FUNCTION_BLOCK STATE_LOGGER_SIMPLE
  {SET_ATTRIBUTE(OpcUa, SERVICE)}
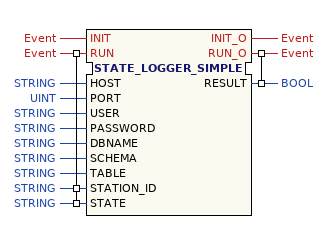
  EVENT_INPUT
    INIT;
    RUN WITH STATION_ID, STATE;
  END_EVENT
  EVENT_OUTPUT
    INIT_O;
    RUN_O WITH RESULT;
  END_EVENT
  VAR_INPUT
    HOST : STRING;
    PORT : UINT;
    USER : STRING;
    PASSWORD : STRING;
    DBNAME : STRING;
    SCHEMA : STRING;
    TABLE : STRING;
    STATION_ID : STRING;
    STATE : STRING;
  END_VAR
  VAR_OUTPUT
    RESULT : BOOL;
  END_VAR
END_FUNCTION_BLOCK
